Yaskawa INFORM job: SKRZYNIA_4640_-90_STOPNI_20BR.JBI

/JOB
//NAME SKRZYNIA_4640_-90_STOPNI_20BR
///FOLDERNAME 02-SKRZYNIE_JOBS
//POS
///NPOS 581,581,0,37,0,0
///TOOL 0
///POSTYPE PULSE
///PULSE
C00000=0,-52280,40443,0,6876,0
C00001=-82314,-24956,17040,-59626,-27382,-6248
C00002=-93910,-8625,17040,-59626,-43355,-6248
C00003=-98846,-1061,-42166,-80308,-57081,16120
C00004=-100452,6057,-48127,-85711,-56704,21322
C00005=-95817,31791,-34187,-84788,-63710,26674
C00006=-95573,33077,-33257,-84645,-64023,26851
C00007=-94315,33778,-32137,-85160,-63467,26714
C00008=-95573,33077,-33257,-84645,-64023,26851
C00009=-94948,31301,-36075,-85235,-63717,27152
C00010=-95573,33077,-33257,-84645,-64023,26851
C00011=-95263,33142,-33256,-84677,-63995,26850
C00012=-95263,33142,-33256,-84677,-63995,26850
C00013=-94230,33719,-32331,-85099,-63538,26735
C00014=-95263,33142,-33256,-84677,-63995,26850
C00015=-94794,31816,-35365,-85120,-63763,27076
C00016=-95263,33142,-33256,-84677,-63995,26850
C00017=-95260,33144,-33256,-84678,-63995,26850
C00018=-95260,33144,-33256,-84678,-63995,26850
C00019=-94260,33701,-32361,-85086,-63552,26738
C00020=-95738,35616,-30155,-83417,-65710,26451
C00021=-94835,31943,-35167,-85080,-63786,27056
C00022=-95260,33144,-33256,-84678,-63995,26850
C00023=-95258,25631,32269,-66559,-75499,2416
C00024=-95258,25631,32269,-66559,-75499,2416
C00025=-94256,26435,33444,-66420,-74940,2208
C00026=-95258,25631,32269,-66559,-75499,2416
C00027=-94857,24030,29962,-66606,-75105,2539
C00028=-95258,25631,32269,-66559,-75499,2416
C00029=-98811,21047,-15512,-99242,-81394,20987
C00030=-98811,21047,-15512,-99242,-81394,20987
C00031=-97856,21592,-14760,-99539,-80803,20995
C00032=-98811,21047,-15512,-99242,-81394,20987
C00033=-98487,19855,-17143,-99373,-81250,21110
C00034=-98811,21047,-15512,-99242,-81394,20987
C00035=-99077,36985,67047,-90824,-74996,11
C00036=-99077,36985,67047,-90824,-74996,11
C00037=-98126,38026,68808,-90519,-74354,-175
C00038=-99077,36985,67047,-90824,-74996,11
C00039=-98675,34279,62554,-90994,-74807,523
C00040=-99077,36985,67047,-90824,-74996,11
C00041=-98046,30065,45001,-99674,-75008,5996
C00042=-96663,27244,32711,-106417,-76052,10001
C00043=-96035,27733,33435,-106407,-75606,10011
C00044=-96663,27244,32711,-106417,-76052,10001
C00045=-96274,25568,30264,-106516,-75947,10234
C00046=-96663,27244,32711,-106417,-76052,10001
C00047=-100395,5963,-6492,-101051,-69866,13942
C00048=-97697,-21147,-29798,-104770,-52931,14344
C00049=-81691,-45027,-49520,-104186,-37412,14105
C00050=-48287,-44591,-17414,-16172,-14532,-25809
C00051=-85348,-13130,13838,-41209,-47455,-8220
C00052=-97998,22495,32685,-69647,-75009,8900
C00053=-98284,29564,37770,-71835,-80250,10571
C00054=-100615,26523,30326,-83718,-79542,3747
C00055=-99528,26746,30653,-83688,-78804,3698
C00056=-98609,27389,31597,-83640,-78189,3601
C00057=-99528,26746,30653,-83688,-78804,3698
C00058=-99278,25562,28929,-83734,-78615,3833
C00059=-99528,26746,30653,-83688,-78804,3698
C00060=-97827,29852,38067,-72347,-79830,10157
C00061=-97362,30289,38867,-71738,-79704,10396
C00062=-96447,31020,39967,-71637,-79179,10220
C00063=-97362,30289,38867,-71738,-79704,10396
C00064=-97069,28896,36765,-71776,-79401,10550
C00065=-97362,30289,38867,-71738,-79704,10396
C00066=-99687,30516,41738,-96594,-77984,-2813
C00067=-99279,34023,49568,-96204,-78485,-4167
C00068=-98297,34881,50932,-96068,-77785,-4257
C00069=-99279,34023,49568,-96204,-78485,-4167
C00070=-98948,32155,46632,-96284,-78364,-3863
C00071=-99279,34023,49568,-96204,-78485,-4167
C00072=-99820,26032,21623,-82067,-78848,-4447
C00073=-99820,26032,21623,-82067,-78848,-4447
C00074=-98898,26645,22513,-82083,-78237,-4546
C00075=-99820,26032,21623,-82067,-78848,-4447
C00076=-99438,24292,19129,-82156,-78552,-4268
C00077=-99820,26032,21623,-82067,-78848,-4447
C00078=-95331,1432,-9864,-84798,-60031,-3557
C00079=-100799,20404,12473,-99797,-78179,2590
C00080=-99814,-4938,-36996,-116444,-71342,12229
C00081=-82620,-30758,-83593,-142203,-62652,21635
C00082=-79591,-62427,-80212,-133576,-39445,13545
C00083=-61872,-66272,-83954,-148251,-32298,21081
C00084=-61872,-49557,-32264,-110357,-15428,1928
C00085=-71091,-37860,2722,-34648,-42002,-27792
C00086=-94097,-13222,20403,-45591,-54273,-19204
C00087=-97363,-23488,-17584,-60839,-44712,-9276
C00088=-98197,-8670,-25604,-81540,-55001,4479
C00089=-99236,18416,3235,-80713,-73731,6125
C00090=-98716,22747,8680,-80557,-75862,6048
C00091=-97982,23215,9333,-80619,-75386,5974
C00092=-98716,22747,8680,-80557,-75862,6048
C00093=-98409,21490,6932,-80649,-75627,6156
C00094=-98716,22747,8680,-80557,-75862,6048
C00095=-100183,29342,35466,-85708,-79719,1114
C00096=-100183,29342,35466,-85708,-79719,1114
C00097=-99011,30198,36753,-85631,-78926,990
C00098=-100183,29342,35466,-85708,-79719,1114
C00099=-99817,27493,32713,-85776,-79458,1347
C00100=-100183,29342,35466,-85708,-79719,1114
C00101=-94729,-288,3800,-87543,-55904,1533
C00102=-77861,-26606,-19905,-76223,-21443,-3330
C00103=-46440,-50562,-32626,1826,-13880,-39178
C00104=-46440,-50562,-32626,1826,-13880,-39178
///LIMIT ON
C00105=-38692,-65390,10180,-18335,3144,1955
///LIMIT OFF
C00106=0,-52280,40443,0,6876,0
C00107=0,-52280,40443,0,6876,0
C00108=0,-43112,23163,32261,-40956,29092
C00109=-48283,-21883,28214,-25170,-26491,48363
C00110=-46664,-3144,58041,-18842,-32105,45325
C00111=-50347,-18571,12268,-49104,-16423,60029
C00112=-52476,-17044,12146,-55476,-16783,62883
C00113=-51467,-16091,12918,-54586,-16145,62570
C00114=-51762,-16375,12685,-54854,-16332,62665
C00115=-53129,-15664,13268,-57063,-16995,63582
C00116=-52557,-17119,12084,-55547,-16837,62908
C00117=-50509,-19000,10610,-51503,-15997,61182
C00118=-52966,-16930,12240,-56194,-17032,63176
C00119=-51879,-15912,13067,-55265,-16346,62852
C00120=-52154,-16175,12851,-55507,-16521,62938
C00121=-53227,-15612,13314,-57215,-17042,63646
C00122=-52966,-16930,12240,-56194,-17032,63176
C00123=-50703,-18403,11066,-52155,-16024,61477
C00124=-52780,-17619,11680,-55562,-17015,62889
C00125=-51306,-16241,12790,-54268,-16084,62435
C00126=-51660,-16583,12512,-54593,-16308,62551
C00127=-53327,-15718,13220,-57282,-17114,63667
C00128=-52780,-17619,11680,-55562,-17015,62889
C00129=-50704,-18401,11069,-52157,-16021,61478
C00130=-53191,-17342,11901,-56260,-17204,63181
C00131=-51773,-16022,12969,-55050,-16305,62760
C00132=-52146,-16378,12679,-55379,-16540,62876
C00133=-53214,-15820,13135,-57085,-17059,63584
C00134=-53002,-17172,12037,-56105,-17083,63128
C00135=-51005,-17995,11387,-52847,-16122,61778
C00136=-52654,-17319,11922,-55560,-16911,62904
C00137=-51372,-16113,12897,-54432,-16099,62508
C00138=-51648,-16379,12679,-54684,-16273,62598
C00139=-52952,-15703,13233,-56807,-16903,63480
C00140=-53323,-17134,12070,-56539,-17248,63304
C00141=-52826,-20105,4812,-63938,-15678,66983
C00142=-52298,-19620,5183,-63681,-15322,66914
C00143=-51076,-18450,6096,-63049,-14499,66733
C00144=-51419,-18785,5831,-63233,-14731,66786
C00145=-52680,-18133,6347,-65138,-15424,67581
C00146=-52924,-19431,7025,-60935,-16175,65505
C00147=-51752,-18759,10786,-53484,-16613,62002
C00148=-52244,-17884,11471,-54682,-16766,62529
C00149=-50303,-16031,12961,-52880,-15542,61887
C00150=-50741,-16464,12607,-53310,-15818,62044
C00151=-52416,-15612,13306,-56135,-16617,63223
C00152=-51898,-18011,11369,-54129,-16600,62301
C00153=-50945,-18019,11363,-52741,-16103,61737
C00154=-51347,-17395,11856,-53690,-16237,62152
C00155=-49990,-16073,12923,-52376,-15383,61677
C00156=-50384,-16465,12603,-52769,-15629,61822
C00157=-52066,-15616,13298,-55654,-16423,63028
C00158=-51792,-17610,11685,-54205,-16494,62350
C00159=-50945,-18019,11363,-52741,-16103,61737
C00160=-50845,-17493,11778,-52895,-15987,61824
C00161=-49521,-16191,12826,-51571,-15155,61341
C00162=-49894,-16567,12520,-51958,-15389,61484
C00163=-51728,-15654,13268,-55171,-16246,62832
C00164=-51082,-17431,11827,-53280,-16102,61986
C00165=-50028,-23690,-6096,-22921,-31075,54538
C00166=-50346,-22995,-5584,-23393,-31002,54768
C00167=-48843,-21430,-4410,-21901,-30270,54078
C00168=-49178,-21788,-4683,-22239,-30433,54235
C00169=-50538,-21100,-4158,-23908,-30654,55032
C00170=-50252,-22811,-5450,-23315,-30936,54734
C00171=-49763,-24818,-32918,-23163,-28604,59699
C00172=-49144,-24298,-32242,-22455,-28505,59304
C00173=-47766,-22458,-30816,-21237,-27774,58615
C00174=-48099,-22913,-31171,-21534,-27949,58786
C00175=-49602,-21997,-30448,-23301,-28174,59772
C00176=-49259,-23869,-32392,-22880,-28141,59533
C00177=-50713,-12366,-58367,-41124,-17813,74400
C00178=-50097,-11438,-57505,-40749,-17495,74109
C00179=-49105,-9842,-55994,-40096,-16991,73614
C00180=-49355,-10250,-56383,-40269,-17116,73742
C00181=-50506,-9357,-55529,-41571,-17503,74586
C00182=-49771,-10920,-57018,-40545,-17327,73951
C00183=-46548,-30139,-39639,-20061,-27197,57955
C00184=-48797,-26670,-6576,-20404,-32539,53259
C00185=-45389,-28224,4312,-35967,-15579,54278
C00186=-40154,-51179,-915,-24203,-8234,36524
C00187=0,-52280,40443,0,6876,0
C00188=0,-52280,40443,0,6876,0
C00189=-2117,-50103,-33543,-4117,45077,85249
C00190=26439,-48928,-33543,-4117,-52362,85249
C00191=26439,-27355,-33543,-41485,-52362,85249
C00192=39218,-24492,-41653,-51934,-39374,86964
C00193=38244,-2284,-24157,-56964,-37300,90090
C00194=26640,586,-20198,-77712,-51919,89712
C00195=26323,460,-20341,-77681,-52125,89737
C00196=25607,3186,-17293,-77585,-52601,89760
C00197=26323,460,-20341,-77681,-52125,89737
C00198=27719,1044,-19697,-77798,-51218,89644
C00199=26640,586,-20198,-77712,-51919,89712
C00200=46457,7101,-11330,-26648,-40775,82885
C00201=47439,8350,-9833,-26106,-40556,82449
C00202=46334,10684,-6981,-26557,-41070,82837
C00203=47439,8350,-9833,-26106,-40556,82449
C00204=48354,9159,-8854,-25603,-40343,82046
C00205=47439,8350,-9833,-26106,-40556,82449
C00206=24760,-3019,-10726,-94610,-54398,89614
C00207=25145,-1220,-8811,-94681,-54143,89655
C00208=24492,1290,-6066,-94601,-54582,89624
C00209=25145,-1220,-8811,-94681,-54143,89655
C00210=26584,-669,-8211,-94866,-53174,89734
C00211=25145,-1220,-8811,-94681,-54143,89655
C00212=14532,-15164,-22494,-92943,-61192,88617
C00213=-33377,-12679,-20251,-90012,-93751,87621
C00214=-32674,-7309,22058,-70557,-98373,80594
C00215=20046,-29908,-41690,-58842,-55822,75080
C00216=46158,10269,-6164,-23128,-46470,70172
C00217=51306,10256,-19432,-23475,-33025,71236
C00218=50386,12004,-17260,-23922,-33430,71616
C00219=51306,10256,-19432,-23475,-33025,71236
C00220=51995,10928,-18601,-23012,-32906,70879
C00221=51306,10256,-19432,-23475,-33025,71236
C00222=50667,8104,-22050,-23976,-33027,71608
C00223=27434,3323,14960,-56922,-57501,78346
C00224=29014,6574,18756,-56344,-56678,77965
C00225=28326,9009,21700,-56459,-57175,78009
C00226=29014,6574,18756,-56344,-56678,77965
C00227=30292,7183,19486,-55908,-55969,77693
C00228=29014,6574,18756,-56344,-56678,77965
C00229=24457,-1296,-8898,-94600,-54606,89622
C00230=24457,-1296,-8898,-94600,-54606,89622
C00231=23939,748,-6672,-94541,-54956,89598
C00232=24457,-1296,-8898,-94600,-54606,89622
C00233=25626,-864,-8432,-94748,-53818,89684
C00234=24457,-1296,-8898,-94600,-54606,89622
C00235=22058,-20035,-26567,-93333,-56013,88551
C00236=-28907,-25632,-31027,-90338,-90583,86609
C00237=-23923,-11573,-19230,-90501,-87328,87840
C00238=-8646,-8251,-7782,-76032,-82054,83740
C00239=42001,26537,64712,-25019,-74648,68382
C00240=42692,25604,59505,-25067,-71864,68798
C00241=42100,27723,62792,-25233,-72628,68820
C00242=42692,25604,59505,-25067,-71864,68798
C00243=43179,26157,60355,-24838,-71882,68629
C00244=42692,25604,59505,-25067,-71864,68798
C00245=42064,17796,48100,-25604,-70267,69397
C00246=28113,-7386,-15136,-95790,-47335,90009
C00247=28228,-6488,-14240,-95859,-47266,90053
C00248=27767,-5044,-12775,-95858,-47588,90072
C00249=28228,-6488,-14240,-95859,-47266,90053
C00250=29468,-5989,-13737,-96077,-46438,90154
C00251=28228,-6488,-14240,-95859,-47266,90053
C00252=51937,664,-7429,-160484,-50080,89770
C00253=52345,1107,-6938,-160727,-50007,89930
C00254=51359,2767,-5080,-160136,-50147,89540
C00255=52345,1107,-6938,-160727,-50007,89930
C00256=53054,1752,-6222,-161147,-49882,90209
C00257=52345,1107,-6938,-160727,-50007,89930
C00258=51937,664,-7429,-160484,-50080,89770
C00259=29691,-10745,-18393,-95770,-46230,89933
C00260=26663,-19279,-25970,-94307,-48104,89008
C00261=29542,-7588,-14846,-100915,-46930,90773
C00262=29616,-6902,-10165,-96183,-45225,84004
C00263=29097,-5391,-8640,-96201,-45588,84023
C00264=29616,-6902,-10165,-96183,-45225,84004
C00265=31098,-6282,-9543,-96410,-44233,84135
C00266=29616,-6902,-10165,-96183,-45225,84004
C00267=7576,-30273,-44451,-97512,-61182,86443
C00268=-18624,-40022,-50597,-93591,-78329,83668
C00269=-32134,-30783,-37092,-96173,-88064,83581
C00270=23774,-1324,-8929,-94512,-55065,89585
C00271=23774,-1324,-8929,-94512,-55065,89585
C00272=23319,517,-6924,-94461,-55372,89567
C00273=23774,-1324,-8929,-94512,-55065,89585
C00274=25077,-853,-8421,-94674,-54188,89653
C00275=23774,-1324,-8929,-94512,-55065,89585
C00276=22107,-1052,28039,-94807,-51389,77849
C00277=19995,-16885,24938,-75612,-39910,62837
C00278=5366,-38499,37552,-33963,-10211,16191
C00279=0,-52280,40443,0,6876,0
C00280=-82314,-24956,17040,-59626,-27382,-6248
C00281=-93910,-8625,17040,-59626,-43355,-6248
C00282=-98846,-1061,-42166,-80308,-57081,16120
C00283=-100452,6057,-48127,-85711,-56704,21322
C00284=-95564,34698,-34234,-85516,-63941,27819
C00285=-94021,36658,-30981,-84167,-64832,27454
C00286=-93851,36773,-30815,-84181,-64812,27439
C00287=-95564,34698,-34234,-85516,-63941,27819
C00288=-96930,32282,-32252,-82595,-65816,26305
C00289=-93901,32995,-31122,-83953,-64436,26132
C00290=-93891,32978,-31150,-83961,-64431,26134
C00291=-96930,32282,-32252,-82595,-65816,26305
C00292=-97719,-4194,-31542,-76086,-54596,10626
C00293=-88377,-34186,-45291,-67238,-52212,2442
C00294=-73560,-62084,7826,-28695,-34737,-3666
C00295=0,-52280,40443,0,6876,0
C00296=0,-52280,40443,0,6876,0
C00297=-2117,-50103,-33543,-4117,45077,85249
C00298=26439,-48928,-33543,-4117,-52362,85249
C00299=26439,-27355,-33543,-41485,-52362,85249
C00300=39218,-24492,-41653,-51934,-39374,86964
C00301=37381,-5106,-22608,-53943,-39515,88347
C00302=38119,-10689,-19379,-70548,-34101,88029
C00303=37906,-14512,-22901,-69984,-34376,87713
C00304=41414,6981,-5927,-33889,-45598,86373
C00305=42289,10624,-1511,-33365,-45508,85956
C00306=42351,10656,-1473,-33340,-45486,85935
C00307=41414,6981,-5927,-33889,-45598,86373
C00308=53221,-12364,-8957,-19277,-47766,73858
C00309=11365,-15171,10010,-30164,-77975,82960
C00310=16156,-38280,11293,-23671,-42998,42040
C00311=11365,-47379,10010,-30164,3063,681
C00312=0,-52280,40443,0,6876,0
C00313=0,-36700,24612,42871,-31823,33862
C00314=-44403,-30110,7154,-24155,-23805,45557
C00315=-51570,-19542,10947,-41619,-21811,53396
C00316=-51570,-17239,16856,-38066,-23574,51584
C00317=-55052,-13712,19754,-43494,-24529,53873
C00318=-55190,-12778,21730,-42693,-25060,53437
C00319=-40431,-28773,9158,-17648,-23273,42875
C00320=0,-36700,24612,42871,-31823,33862
C00321=0,-52280,40443,0,6876,0
C00322=0,-52280,40443,0,6876,0
C00323=-73560,-62084,7826,-28695,-34737,-3666
C00324=-88377,-34186,-45291,-67238,-52212,2442
C00325=-99860,-8392,-35780,-75647,-56000,10650
C00326=-100432,21324,12575,-83706,-77956,7498
C00327=-100432,21324,12575,-83706,-77956,7498
C00328=-97477,24790,17443,-83584,-77881,7143
C00329=-97548,25214,18044,-83537,-78171,7107
C00330=-100432,21324,12575,-83706,-77956,7498
C00331=-100473,21504,12824,-83696,-77986,7482
C00332=-97708,25565,18549,-83502,-78342,7077
C00333=-97720,26100,19317,-83456,-78605,7025
C00334=-100432,21324,12575,-83706,-77956,7498
C00335=-98403,3681,-8965,-86029,-63956,7946
C00336=-99524,-11453,-5366,-86029,-50962,7946
C00337=-93426,-21174,-16075,-79197,-62083,2349
C00338=-58820,-39124,10926,-53325,-41870,-3759
C00339=0,-52280,40443,0,6876,0
C00340=-37281,-50778,-9546,-79570,-75313,71156
C00341=-21038,-23698,-30323,-82948,-81132,85647
C00342=-21230,-24252,-33397,-84866,-81311,86227
C00343=26224,-11477,-22521,-89106,-49066,87170
C00344=30473,789,4724,-68168,-47848,79016
C00345=30460,-1091,-3608,-71823,-46530,81583
C00346=26224,-11477,-22521,-89106,-49066,87170
C00347=1250,-26379,-34995,-85812,-66036,85728
C00348=-29373,-17697,-13794,-84248,-87305,82376
C00349=-12562,-22815,-22029,-52123,-75138,85349
C00350=41964,2536,-13642,-34848,-42769,74522
C00351=37974,4101,-26304,-58477,-36842,84551
C00352=37992,4823,-31618,-63468,-34913,87461
C00353=41439,5489,-14791,-37032,-40569,75962
C00354=38833,-3286,10682,-41231,-51577,69207
C00355=-9276,-22918,-17698,-90837,-69000,78700
C00356=-8172,-56778,-49528,-75726,-40055,75711
C00357=-3982,-61001,-53003,-69042,-33087,73336
C00358=37287,-55159,35520,-2191,5667,2084
C00359=0,-52280,40443,0,6876,0
C00360=0,-36700,24612,42871,-31823,33862
C00361=-44403,-30110,7154,-24155,-23805,45557
C00362=-44403,-30110,7154,-24155,-23805,45557
C00363=-42101,-12213,25656,-103795,-5192,78630
C00364=-46259,-8171,27719,-110365,-8144,81138
C00365=-49067,-3914,32085,-108223,-9817,79727
C00366=-55938,-2414,24284,-132193,-25662,89374
C00367=-55845,-2055,25408,-131547,-25258,89050
C00368=-56934,-15752,2926,-132390,-27589,90381
C00369=-47073,-34549,9488,-27883,-30316,51458
C00370=0,-52280,40443,0,6876,0
C00371=0,-52280,40443,0,6876,0
C00372=-73560,-62084,7826,-28695,-34737,-3666
C00373=-96366,-17217,16860,-56620,-71703,-18245
C00374=-98152,-14905,2044,-65675,-67485,-3494
C00375=-100467,-7393,-15195,-81625,-60158,6002
C00376=-99336,18440,8642,-84276,-74234,7647
C00377=-99336,18440,8642,-84276,-74234,7647
C00378=-97907,25479,18429,-83510,-78268,7080
C00379=-97774,25771,18838,-83486,-78362,7054
C00380=-99336,18440,8642,-84276,-74234,7647
C00381=-88887,-29565,-44699,-91336,-36715,8429
C00382=-85230,-48302,-58733,-86716,-36654,5475
C00383=-60204,-59872,-73451,-117647,-17639,18840
C00384=-37721,-67612,11381,-1325,-438,-7850
C00385=0,-52280,40443,0,6876,0
C00386=37287,-55159,35520,-2191,5667,2084
C00387=40042,-68802,-18337,-47708,-19461,45384
C00388=16481,-63411,-38742,-86271,-37962,67106
C00389=28646,-23138,-32952,-89786,-42552,85395
C00390=38882,-16596,-17625,-44304,-41043,72768
C00391=40930,-6862,-13364,-47045,-37020,74415
C00392=41744,-3361,-9781,-46774,-36492,74231
C00393=41678,-4243,-16493,-50979,-33997,76666
C00394=40930,-6862,-13364,-47045,-37020,74415
C00395=38882,-16596,-17625,-44304,-41043,72768
C00396=28646,-23138,-32952,-89786,-42552,85395
C00397=29905,-15291,-26411,-91102,-43435,86304
C00398=31540,-7654,-19248,-92177,-42391,86919
C00399=31445,-8095,-22888,-97196,-43117,89457
C00400=29637,-16450,-35189,-96198,-44206,89682
C00401=-7164,-46429,-55577,-86274,-68578,84143
C00402=40042,-68802,-18337,-47708,-19461,45384
C00403=37287,-55159,35520,-2191,5667,2084
C00404=0,-52280,40443,0,6876,0
C00405=-37164,-60659,6466,-13301,-5027,19773
C00406=-45362,-39990,2831,-27538,-17767,40935
C00407=-57189,-26834,-7130,-38780,-31731,51561
C00408=-55974,-20661,-3180,-39617,-29741,52134
C00409=-55991,-28453,-45977,-64163,-20900,63765
C00410=-57189,-26834,-7130,-38780,-31731,51561
C00411=-41180,-61187,4729,-17280,-8498,23442
C00412=0,-52280,40443,0,6876,0
C00413=0,-52280,40443,0,6876,0
C00414=-43180,-50572,-20637,-6552,-29302,-38834
C00415=-79425,-37128,-15462,-51820,-35721,-18807
C00416=-93702,-21743,-5664,-65079,-41536,-12324
C00417=-95468,-3718,3432,-57810,-54196,-8058
C00418=-98195,18244,29331,-65465,-72367,-4307
C00419=-96728,36447,56610,-70336,-82085,-4645
C00420=-96821,31985,42520,-71106,-80277,-1800
C00421=-99571,23446,29328,-71481,-76214,-993
C00422=-98368,-15155,-15320,-68503,-52006,-4003
C00423=-90196,-30440,-22000,-63685,-45526,-9297
C00424=-44920,-50063,-20090,-8739,-29356,-37564
C00425=-37721,-67612,11381,-1325,-438,-7850
C00426=0,-52280,40443,0,6876,0
C00427=40043,-68802,-18337,-47706,-19461,45383
C00428=27078,-46675,7729,-35821,-60236,53359
C00429=37661,6027,34279,-36092,-58837,68690
C00430=38848,9668,32452,-36978,-55195,69693
C00431=45203,15557,41040,-24527,-60177,66840
C00432=37661,2340,23735,-37788,-55306,70200
C00433=22173,-30639,7984,-58136,-45615,60133
C00434=37287,-55159,35520,-2191,5667,2084
C00435=0,-52280,40443,0,6876,0
C00436=-23708,-46776,23536,-16027,-4787,19738
C00437=-50917,-40459,4132,-34421,-18173,42391
C00438=-54964,-26842,8528,-44141,-23181,52038
C00439=-51719,-20944,8196,-48593,-18539,54728
C00440=-53338,-16066,12564,-52314,-18938,56375
C00441=-53668,-14237,17353,-48629,-20286,54493
C00442=-18010,-41727,-5437,24633,-20435,23511
C00443=-41180,-61187,4729,-17280,-8498,23442
C00444=0,-52280,40443,0,6876,0
C00445=0,-52280,40443,0,6876,0
C00446=-37721,-67612,11381,-1325,-438,-7850
C00447=-43180,-50572,-20637,-6552,-29302,-38834
C00448=-79425,-37128,-15462,-51820,-35721,-18807
C00449=-92377,-33385,-41303,-83059,-36844,-1354
C00450=-98043,-4314,-16897,-86107,-58749,2387
C00451=-99186,-1007,-13605,-90357,-63007,3800
C00452=-99448,23410,16807,-87478,-77479,2357
C00453=-98529,24761,18725,-87324,-78429,2215
C00454=-98419,25196,20150,-87169,-78534,1864
C00455=-99450,-173,-12700,-90327,-63185,3798
C00456=-99875,3426,-9244,-98609,-66692,6315
C00457=-99431,-3293,-16601,-99643,-62713,6757
C00458=-92822,-26306,-37175,-103295,-43881,7703
C00459=-68601,-52593,-52127,-95725,-25602,3235
C00460=-80632,-38079,-20908,-64053,-45216,-12949
C00461=-43180,-50572,-20637,-6552,-29302,-38834
C00462=-37721,-67612,11381,-1325,-438,-7850
C00463=0,-52280,40443,0,6876,0
C00464=-7830,-25136,17099,-55306,-64068,52084
C00465=34592,-23156,18291,-29932,-45204,43222
C00466=27626,-5609,7480,-74303,-46810,69713
C00467=30162,-7263,-3756,-79871,-43922,73611
C00468=30945,-3557,12,-79972,-43367,73694
C00469=30934,-3652,-86,-79966,-43372,73693
C00470=29106,-7674,-4162,-79972,-44640,73655
C00471=-2837,-32019,-23857,-80741,-66785,72567
C00472=9534,-43450,13514,-26959,-29486,38723
C00473=22834,-59963,22946,-6692,-2150,9612
C00474=0,-52280,40443,0,6876,0
C00475=-23708,-46776,23536,-16027,-4787,19738
C00476=-50917,-40459,4132,-34421,-18173,42391
C00477=-51059,-36587,4608,-36647,-19418,45358
C00478=-50113,-22729,10834,-36393,-23396,50963
C00479=-58003,-17258,7975,-66354,-22196,69294
C00480=-57660,-15851,11780,-61832,-22634,66694
C00481=-50113,-22729,10834,-36393,-23396,50963
C00482=-45969,-44671,-42317,80322,10570,10889
C00483=-31285,-69981,-10849,-7246,-6842,20992
C00484=0,-52280,40443,0,6876,0
C00485=-37721,-67612,11381,-1325,-438,-7850
C00486=-43180,-50572,-20637,-6552,-29302,-38834
C00487=-79425,-37128,-15462,-51820,-35721,-18807
C00488=-92377,-33385,-41303,-83059,-36844,-1354
C00489=-97955,-4566,-17156,-86109,-58691,2381
C00490=-98763,-4191,-27333,-97091,-62203,7437
C00491=-100541,17285,32324,-96596,-68502,-4435
C00492=-99163,31411,54049,-96228,-73919,-6997
C00493=-97653,31369,46884,-97568,-75920,-4787
C00494=-97653,34871,57346,-96543,-75121,-6929
C00495=-98792,6748,2422,-99606,-66785,1957
C00496=-99852,25442,19906,-82977,-78439,1439
C00497=-97669,24909,7904,-99153,-81388,7704
C00498=-97669,24909,7904,-99153,-81388,7704
C00499=-99984,22604,5279,-91306,-78940,6306
C00500=-98813,-5502,-22210,-93134,-60245,5727
C00501=-97559,-25159,-36085,-93407,-46496,3918
C00502=-68601,-52593,-52127,-95725,-25602,3235
C00503=-80632,-38079,-20908,-64053,-45216,-12949
C00504=-43180,-50572,-20637,-6552,-29302,-38834
C00505=-37721,-67612,11381,-1325,-438,-7850
C00506=54026,-30203,28811,7745,-28969,5087
C00507=55906,-29650,27841,6704,-28568,42061
C00508=3910,-49110,-20873,-64325,-51391,71742
C00509=9596,-41005,-15480,-61992,-50741,70573
C00510=34629,-5327,8260,-51720,-47880,65426
C00511=35679,2837,17551,-51053,-47466,65038
C00512=35689,-56,7549,-54586,-44718,67469
C00513=34629,-5327,8260,-51720,-47880,65426
C00514=9596,-41005,-15480,-61992,-50741,70573
C00515=29660,-4584,-26917,-122917,-59269,85605
C00516=30458,-1431,-23593,-123278,-58903,85810
C00517=32051,-581,-21149,-126899,-58917,85995
C00518=28378,-5181,-30467,-124970,-61925,86269
C00519=9596,-41005,-15480,-61992,-50741,70573
C00520=4124,-42500,-16101,-63937,-54198,71061
C00521=22834,-59963,22946,-6692,-2150,9612
C00522=0,-52280,40443,0,6876,0
C00523=-44101,-76445,-48847,-15697,-17168,40457
C00524=-48984,-30078,-36716,-21434,-29637,58750
C00525=-50484,-13386,-55713,-36158,-19724,71897
C00526=-50484,-10141,-52609,-36672,-19476,72159
C00527=-57834,15023,-57436,-77444,-21310,89314
C00528=-50484,-13386,-55713,-36158,-19724,71897
C00529=-49763,-25421,-36239,-24565,-26935,60445
C00530=-50529,-22709,-3778,-22940,-31995,54502
C00531=-45389,-28224,4312,-35967,-15579,54278
C00532=-40154,-51179,-915,-24203,-8234,36524
C00533=0,-52280,40443,0,6876,0
C00534=0,-52280,40443,0,6876,0
C00535=-37721,-67612,11381,-1325,-438,-7850
C00536=-43180,-50572,-20637,-6552,-29302,-38834
C00537=-43180,-50572,-20637,-6552,-29302,-38834
C00538=-91571,-17240,10754,-52986,-45776,-17944
C00539=-85565,-2479,24798,-50710,-47830,-17652
C00540=-84901,-1641,24348,-52361,-47087,-17020
C00541=-100018,24469,26124,-84922,-77496,-993
C00542=-98221,24171,26084,-84881,-76275,-1110
C00543=-97925,23780,23736,-81145,-76027,-1196
C00544=-96886,22779,17134,-75074,-74614,-730
C00545=-96886,21697,9827,-76119,-73731,1247
C00546=-99355,23812,23162,-76774,-76908,-1703
C00547=-99772,22813,18672,-85812,-76963,849
C00548=-98588,26860,21106,-87462,-79585,-1754
C00549=-98621,27173,20618,-87985,-79896,-2348
C00550=-99360,20896,24116,-84704,-74336,-1671
C00551=-89794,-9992,-7341,-81590,-44258,-3681
C00552=-98228,-14972,-11291,-81392,-49231,-4002
C00553=-98228,-7428,13566,-72439,-51372,-10695
C00554=-68865,-35989,-5252,-49829,-38105,-21179
C00555=-40763,-44623,-7750,-16844,-36810,-34738
C00556=0,-52278,40443,-31822,-65283,46097
C00557=7820,3000,44222,-77356,-66876,70486
C00558=23103,22769,71034,-65639,-61603,67373
C00559=25078,30713,84198,-63240,-61811,65668
C00560=25008,30264,83410,-63369,-61766,65773
C00561=23103,22769,71034,-65639,-61603,67373
C00562=23103,22769,71034,-65639,-61603,67373
C00563=25078,30713,84198,-63240,-61811,65668
C00564=25008,30264,83410,-63369,-61766,65773
C00565=23103,22769,71034,-65639,-61603,67373
C00566=-3014,-20441,-7349,-104591,-68614,79454
C00567=-3014,-20441,-7349,-104591,-68614,79454
C00568=-13238,-21720,-1359,-93359,-59492,72612
C00569=10261,-46634,14475,-36899,-22136,31570
C00570=22834,-59963,22946,-6692,-2150,9612
C00571=0,-52280,40443,0,6876,0
C00572=-23708,-46776,23536,-16027,-4787,19738
C00573=-50917,-40459,4132,-34421,-18173,42391
C00574=-49876,-21948,7530,-68838,-10324,59148
C00575=-46721,-18942,9765,-68167,-8197,59205
C00576=-47734,-15041,12007,-78406,-8476,63945
C00577=-48173,-14749,12492,-78097,-8776,63748
C00578=-42573,-24036,4541,-56448,-5917,54155
C00579=-31287,-69981,-10850,-7253,-6843,20996
C00580=0,-52280,40443,0,6876,0
BC00000=455888
BC00001=445130
BC00002=445130
BC00003=445130
BC00004=445130
BC00005=467179
BC00006=468227
BC00007=468227
BC00008=468227
BC00009=468227
BC00010=468227
BC00011=514421
BC00012=514421
BC00013=514421
BC00014=514421
BC00015=514421
BC00016=514421
BC00017=560588
BC00018=560588
BC00019=560588
BC00020=560588
BC00021=560588
BC00022=560588
BC00023=536404
BC00024=536404
BC00025=536404
BC00026=536404
BC00027=536404
BC00028=536404
BC00029=582458
BC00030=582458
BC00031=582458
BC00032=582458
BC00033=582458
BC00034=582458
BC00035=581206
BC00036=581206
BC00037=581206
BC00038=581206
BC00039=581206
BC00040=581206
BC00041=608443
BC00042=608308
BC00043=608308
BC00044=608308
BC00045=608308
BC00046=608308
BC00047=554082
BC00048=550688
BC00049=540680
BC00050=699121
BC00051=714117
BC00052=772491
BC00053=770398
BC00054=668005
BC00055=668005
BC00056=668005
BC00057=668005
BC00058=668005
BC00059=668005
BC00060=765624
BC00061=770398
BC00062=770398
BC00063=770398
BC00064=770398
BC00065=770398
BC00066=795066
BC00067=795066
BC00068=795066
BC00069=795066
BC00070=795066
BC00071=795066
BC00072=855510
BC00073=855510
BC00074=855510
BC00075=855510
BC00076=855510
BC00077=855510
BC00078=855510
BC00079=800260
BC00080=807414
BC00081=829241
BC00082=831883
BC00083=872244
BC00084=872244
BC00085=900921
BC00086=897901
BC00087=922181
BC00088=915260
BC00089=906767
BC00090=899976
BC00091=899976
BC00092=899976
BC00093=899976
BC00094=899976
BC00095=940845
BC00096=940845
BC00097=940845
BC00098=940845
BC00099=940845
BC00100=940845
BC00101=861557
BC00102=891834
BC00103=895420
BC00104=874556
BC00105=799329
BC00106=750352
BC00107=750350
BC00108=750352
BC00109=858258
BC00110=858258
BC00111=887560
BC00112=953382
BC00113=953382
BC00114=953382
BC00115=953382
BC00116=953382
BC00117=888056
BC00118=888056
BC00119=888056
BC00120=888056
BC00121=888056
BC00122=888056
BC00123=830714
BC00124=830714
BC00125=830714
BC00126=830714
BC00127=830714
BC00128=830714
BC00129=764829
BC00130=764829
BC00131=764829
BC00132=764829
BC00133=764829
BC00134=764829
BC00135=707174
BC00136=707174
BC00137=707174
BC00138=707174
BC00139=707174
BC00140=707174
BC00141=642071
BC00142=642071
BC00143=642071
BC00144=642071
BC00145=642071
BC00146=642071
BC00147=584746
BC00148=584746
BC00149=584746
BC00150=584746
BC00151=584746
BC00152=584746
BC00153=519232
BC00154=519232
BC00155=519232
BC00156=519232
BC00157=519232
BC00158=519232
BC00159=461813
BC00160=461813
BC00161=461813
BC00162=461813
BC00163=461813
BC00164=461813
BC00165=459544
BC00166=459544
BC00167=459544
BC00168=459544
BC00169=459544
BC00170=459544
BC00171=459544
BC00172=459544
BC00173=459544
BC00174=459544
BC00175=459544
BC00176=459544
BC00177=459544
BC00178=459544
BC00179=459544
BC00180=459544
BC00181=459544
BC00182=459544
BC00183=459544
BC00184=459544
BC00185=459540
BC00186=533216
BC00187=533216
BC00188=492150
BC00189=423885
BC00190=423885
BC00191=423885
BC00192=423885
BC00193=423885
BC00194=423882
BC00195=423882
BC00196=423882
BC00197=423882
BC00198=423882
BC00199=423882
BC00200=517447
BC00201=516208
BC00202=516208
BC00203=516208
BC00204=516208
BC00205=516208
BC00206=462401
BC00207=462401
BC00208=462401
BC00209=462401
BC00210=462401
BC00211=462401
BC00212=462401
BC00213=462401
BC00214=581968
BC00215=647467
BC00216=647467
BC00217=647467
BC00218=647467
BC00219=647467
BC00220=647467
BC00221=647467
BC00222=647467
BC00223=600589
BC00224=600589
BC00225=600589
BC00226=600589
BC00227=600589
BC00228=600589
BC00229=646713
BC00230=646713
BC00231=646713
BC00232=646713
BC00233=646713
BC00234=646713
BC00235=646713
BC00236=646713
BC00237=703926
BC00238=764819
BC00239=734650
BC00240=734650
BC00241=734650
BC00242=734650
BC00243=734650
BC00244=734650
BC00245=734650
BC00246=762000
BC00247=762000
BC00248=762000
BC00249=762000
BC00250=762000
BC00251=762000
BC00252=768744
BC00253=768744
BC00254=768744
BC00255=768744
BC00256=768744
BC00257=768744
BC00258=768744
BC00259=762000
BC00260=762000
BC00261=869424
BC00262=869424
BC00263=869424
BC00264=869424
BC00265=869424
BC00266=869424
BC00267=869424
BC00268=869424
BC00269=983898
BC00270=992364
BC00271=992364
BC00272=992364
BC00273=992364
BC00274=992364
BC00275=992364
BC00276=927243
BC00277=910363
BC00278=716208
BC00279=458496
BC00280=445130
BC00281=445130
BC00282=445130
BC00283=445130
BC00284=475938
BC00285=475917
BC00286=468314
BC00287=475938
BC00288=515329
BC00289=515329
BC00290=508301
BC00291=515329
BC00292=542207
BC00293=542207
BC00294=542207
BC00295=542207
BC00296=492150
BC00297=423885
BC00298=423885
BC00299=423885
BC00300=423885
BC00301=418215
BC00302=406365
BC00303=406365
BC00304=507950
BC00305=507950
BC00306=500226
BC00307=507950
BC00308=493160
BC00309=493160
BC00310=493160
BC00311=493160
BC00312=493160
BC00313=582810
BC00314=655182
BC00315=714528
BC00316=712780
BC00317=712780
BC00318=773753
BC00319=773753
BC00320=582810
BC00321=540924
BC00322=542207
BC00323=542207
BC00324=542207
BC00325=590944
BC00326=543764
BC00327=459277
BC00328=459277
BC00329=451665
BC00330=459277
BC00331=520748
BC00332=520748
BC00333=528295
BC00334=520748
BC00335=524597
BC00336=524597
BC00337=555662
BC00338=584417
BC00339=584417
BC00340=542360
BC00341=599440
BC00342=482963
BC00343=482963
BC00344=482963
BC00345=482963
BC00346=482963
BC00347=482963
BC00348=482963
BC00349=633179
BC00350=633182
BC00351=633182
BC00352=633182
BC00353=633182
BC00354=590162
BC00355=577838
BC00356=565789
BC00357=612529
BC00358=620193
BC00359=620193
BC00360=812803
BC00361=887783
BC00362=927066
BC00363=893694
BC00364=914884
BC00365=914884
BC00366=943670
BC00367=973194
BC00368=945981
BC00369=853059
BC00370=542207
BC00371=542207
BC00372=513519
BC00373=556866
BC00374=576802
BC00375=590944
BC00376=571989
BC00377=566860
BC00378=566866
BC00379=572997
BC00380=566860
BC00381=580682
BC00382=599892
BC00383=633159
BC00384=733103
BC00385=733103
BC00386=620193
BC00387=620193
BC00388=625652
BC00389=635598
BC00390=635598
BC00391=635598
BC00392=635598
BC00393=635598
BC00394=635598
BC00395=635598
BC00396=635598
BC00397=658627
BC00398=658630
BC00399=665879
BC00400=658627
BC00401=658627
BC00402=620193
BC00403=620193
BC00404=620193
BC00405=561542
BC00406=498768
BC00407=452071
BC00408=452071
BC00409=452071
BC00410=452071
BC00411=524165
BC00412=524165
BC00413=733103
BC00414=733103
BC00415=646139
BC00416=646133
BC00417=684512
BC00418=682982
BC00419=682982
BC00420=682982
BC00421=682982
BC00422=682236
BC00423=687704
BC00424=698572
BC00425=733103
BC00426=733103
BC00427=667407
BC00428=721208
BC00429=721208
BC00430=721208
BC00431=727232
BC00432=730010
BC00433=686453
BC00434=620193
BC00435=620193
BC00436=576077
BC00437=541793
BC00438=580754
BC00439=589556
BC00440=589433
BC00441=647350
BC00442=649294
BC00443=561088
BC00444=547800
BC00445=733103
BC00446=733103
BC00447=733103
BC00448=733103
BC00449=733103
BC00450=733103
BC00451=740531
BC00452=740531
BC00453=740531
BC00454=745553
BC00455=740531
BC00456=750469
BC00457=750469
BC00458=750469
BC00459=750469
BC00460=783373
BC00461=795297
BC00462=733103
BC00463=733103
BC00464=727492
BC00465=727492
BC00466=759331
BC00467=759331
BC00468=759331
BC00469=766564
BC00470=759331
BC00471=759331
BC00472=672725
BC00473=672725
BC00474=672725
BC00475=766882
BC00476=791101
BC00477=802867
BC00478=836517
BC00479=836517
BC00480=895002
BC00481=836517
BC00482=798026
BC00483=767805
BC00484=733103
BC00485=733103
BC00486=733103
BC00487=733103
BC00488=733103
BC00489=733103
BC00490=815683
BC00491=777789
BC00492=777789
BC00493=784987
BC00494=784987
BC00495=788909
BC00496=855225
BC00497=846870
BC00498=855158
BC00499=855225
BC00500=811096
BC00501=804355
BC00502=750469
BC00503=783373
BC00504=795297
BC00505=733103
BC00506=762701
BC00507=765633
BC00508=830967
BC00509=835024
BC00510=852883
BC00511=852883
BC00512=852883
BC00513=852883
BC00514=835024
BC00515=861491
BC00516=861491
BC00517=861491
BC00518=861491
BC00519=835024
BC00520=835024
BC00521=672725
BC00522=672725
BC00523=528256
BC00524=459544
BC00525=459544
BC00526=459546
BC00527=459544
BC00528=459544
BC00529=459544
BC00530=459544
BC00531=459540
BC00532=533216
BC00533=533216
BC00534=733103
BC00535=733103
BC00536=854587
BC00537=886854
BC00538=885269
BC00539=885269
BC00540=923671
BC00541=946274
BC00542=946274
BC00543=946274
BC00544=907872
BC00545=907872
BC00546=907872
BC00547=970029
BC00548=970060
BC00549=977448
BC00550=970029
BC00551=911970
BC00552=906746
BC00553=883967
BC00554=913920
BC00555=863532
BC00556=921533
BC00557=921533
BC00558=946591
BC00559=946591
BC00560=953713
BC00561=946591
BC00562=997282
BC00563=997282
BC00564=1004404
BC00565=997282
BC00566=1013986
BC00567=963295
BC00568=908449
BC00569=754884
BC00570=672725
BC00571=672725
BC00572=562340
BC00573=452362
BC00574=452362
BC00575=452362
BC00576=452362
BC00577=512870
BC00578=511886
BC00579=742282
BC00580=742282
///POSTYPE BASE
///RECTAN
///RCONF 1,0,0,0,0,0,0,0,0,0,0,0,0,0,0,0,0,0,0,0,0,0,0,0
P00006=0.000,0.000,0.000,0.0000,0.0000,0.0000
P00300=-0.036,-1.505,2.318,0.0000,0.0000,0.0000
P00301=0.046,-2.112,7.779,0.0000,0.0000,0.0000
P00302=-0.180,-2.409,6.326,0.0000,0.0000,0.0000
///RCONF 0,0,0,0,0,0,0,0,0,0,0,0,0,0,0,0,0,0,0,0,0,0,0,0
P00303=-0.004,-1.437,-4.584,0.0000,0.0000,0.0000
P00304=0.028,-1.666,-4.234,0.0000,0.0000,0.0000
P00305=-0.003,-1.920,-3.501,0.0000,0.0000,0.0000
P00306=0.015,-2.252,-3.054,0.0000,0.0000,0.0000
P00307=0.019,-2.151,-5.077,0.0000,0.0000,0.0000
P00308=-0.003,-2.092,-4.888,0.0000,0.0000,0.0000
P00309=-0.040,-2.205,-4.992,0.0000,0.0000,0.0000
P00310=-0.006,-2.490,-5.925,0.0000,0.0000,0.0000
P00311=-0.007,-2.079,-5.307,0.0000,0.0000,0.0000
P00350=11.519,-0.008,1.149,0.0000,0.0000,0.0000
P00351=13.563,-0.027,-0.653,0.0000,0.0000,0.0000
P00352=13.252,-0.027,-0.827,0.0000,0.0000,0.0000
P00353=10.971,-0.082,0.776,0.0000,0.0000,0.0000
P00354=-0.024,2.508,-1.824,0.0000,0.0000,0.0000
P00355=-0.001,2.528,-1.131,0.0000,0.0000,0.0000
P00356=-0.034,2.921,-0.262,0.0000,0.0000,0.0000
P00357=0.003,3.386,-0.091,0.0000,0.0000,0.0000
P00358=0.014,3.037,-0.020,0.0000,0.0000,0.0000
P00359=-0.005,2.731,0.912,0.0000,0.0000,0.0000
P00360=-0.011,3.412,0.438,0.0000,0.0000,0.0000
P00361=0.018,3.050,1.253,0.0000,0.0000,0.0000
P00400=5.920,-3.503,-0.024,0.0000,0.0000,0.0000
P00401=3.430,-0.021,1.131,0.0000,0.0000,0.0000
P00402=-0.253,1.107,3.062,0.0000,0.0000,0.0000
P00403=-3.666,-0.015,5.328,0.0000,0.0000,0.0000
///RCONF 1,0,0,0,0,0,0,0,0,0,0,0,0,0,0,0,0,0,0,0,0,0,0,0
P00404=0.029,4.189,-1.030,0.0000,0.0000,0.0000
///RCONF 0,0,0,0,0,0,0,0,0,0,0,0,0,0,0,0,0,0,0,0,0,0,0,0
P00405=2.420,0.007,1.427,0.0000,0.0000,0.0000
P00406=3.513,-0.022,0.429,0.0000,0.0000,0.0000
///RCONF 1,0,0,0,1,0,0,0,0,0,0,0,0,0,0,0,0,0,0,0,0,0,0,0
P00407=-0.029,2.348,-1.469,0.0000,0.0000,0.0000
P00408=0.010,1.346,-1.479,0.0000,0.0000,0.0000
///RCONF 1,0,0,0,0,0,0,0,0,0,0,0,0,0,0,0,0,0,0,0,0,0,0,0
P00409=-0.026,2.090,-1.483,0.0000,0.0000,0.0000
P00410=0.001,4.491,-0.583,0.0000,0.0000,0.0000
///RCONF 1,0,0,0,1,0,0,0,0,0,0,0,0,0,0,0,0,0,0,0,0,0,0,0
P00411=-0.015,3.627,0.872,0.0000,0.0000,0.0000
//INST
///DATE 2024/11/22 15:59
///ATTR SC,RW
///GROUP1 RB1,BS1
NOP
CALL JOB:MOVE_INTO_TUNNEL
MOVJ C00000 BC00000 VJ=30.00
MOVJ C00001 BC00001 VJ=30.00
MOVJ C00002 BC00002 VJ=30.00
MOVL C00003 BC00003 V=500.0
MOVJ C00004 BC00004 VJ=20.00
'------------------------
'W65.3
'------------------------
MOVL C00005 BC00005 V=333.3
MOVL C00006 BC00006 V=166.7 PL=0
REFP 3 C00007 BC00007
CALL JOB:SEARCH-R1
SET P0300 P0006
SFTON P0300
MOVL C00008 BC00008 V=66.7 PL=0
REFP 3 C00009 BC00009
CALL JOB:SEARCH-R1
SET P0300 P0006
SFTON P0300
MOVL C00010 BC00010 V=66.7 PL=0
SFTOF
'------------------------
'W65.5
'------------------------
MOVL C00011 BC00011 V=500.0
MOVL C00012 BC00012 V=166.7 PL=0
REFP 3 C00013 BC00013
CALL JOB:SEARCH-R1
SET P0301 P0006
SFTON P0301
MOVL C00014 BC00014 V=166.7 PL=0
REFP 3 C00015 BC00015
CALL JOB:SEARCH-R1
SET P0301 P0006
SFTON P0301
MOVL C00016 BC00016 V=166.7 PL=0
SFTOF
'------------------------
'W65.7
'------------------------
MOVL C00017 BC00017 V=500.0
MOVL C00018 BC00018 V=166.7 PL=0
REFP 3 C00019 BC00019
CALL JOB:SEARCH-R1
SET P0302 P0006
SFTON P0302
MOVL C00020 BC00020 V=166.7 PL=0
REFP 3 C00021 BC00021
CALL JOB:SEARCH-R1
SET P0302 P0006
SFTON P0302
MOVL C00022 BC00022 V=166.7 PL=0
SFTOF
'------------------------
'W65.10
'------------------------
MOVL C00023 BC00023 V=500.0
MOVL C00024 BC00024 V=166.7 PL=0
REFP 3 C00025 BC00025
CALL JOB:SEARCH-R1
SET P0303 P0006
SFTON P0303
MOVL C00026 BC00026 V=166.7 PL=0
REFP 3 C00027 BC00027
CALL JOB:SEARCH-R1
SET P0303 P0006
SFTON P0303
MOVL C00028 BC00028 V=166.7 PL=0
SFTOF
'------------------------
'W65.12
'------------------------
MOVL C00029 BC00029 V=500.0
MOVL C00030 BC00030 V=166.7 PL=0
REFP 3 C00031 BC00031
CALL JOB:SEARCH-R1
SET P0304 P0006
SFTON P0304
MOVL C00032 BC00032 V=166.7 PL=0
REFP 3 C00033 BC00033
CALL JOB:SEARCH-R1
SET P0304 P0006
SFTON P0304
MOVL C00034 BC00034 V=166.7 PL=0
SFTOF
'------------------------
'W65.15
'------------------------
COMM MOVL C00035 BC00035 V=333.3
COMM MOVL C00036 BC00036 V=166.7 PL=0
COMM REFP 3 C00037 BC00037
COMM CALL JOB:SEARCH-R1
COMM SET P0305 P0006
COMM SFTON P0305
COMM MOVL C00038 BC00038 V=166.7 PL=0
COMM REFP 3 C00039 BC00039
COMM CALL JOB:SEARCH-R1
COMM SET P0305 P0006
COMM SFTON P0305
COMM MOVL C00040 BC00040 V=166.7 PL=0
COMM SFTOF
COMM '------------------------
COMM 'W65.17
COMM '------------------------
COMM MOVL C00041 BC00041 V=333.3
COMM MOVL C00042 BC00042 V=166.7 PL=0
COMM REFP 3 C00043 BC00043
COMM CALL JOB:SEARCH-R1
COMM SET P0306 P0006
COMM SFTON P0306
COMM MOVL C00044 BC00044 V=166.7 PL=0
COMM REFP 3 C00045 BC00045
COMM CALL JOB:SEARCH-R1
COMM SET P0306 P0006
COMM SFTON P0306
COMM MOVL C00046 BC00046 V=166.7 PL=0
COMM SFTOF
MOVL C00047 BC00047 V=333.3
MOVL C00048 BC00048 V=500.0
MOVL C00049 BC00049 V=500.0
MOVJ C00050 BC00050 VJ=50.00
MOVL C00051 BC00051 V=500.0
MOVL C00052 BC00052 V=500.0
'------------------------
'W65.20
'------------------------
MOVL C00053 BC00053 V=166.7
MOVL C00054 BC00054 V=416.7
MOVL C00055 BC00055 V=166.7 PL=0
REFP 3 C00056 BC00056
CALL JOB:SEARCH-R1
SET P0306 P0006
SFTON P0306
MOVL C00057 BC00057 V=166.7 PL=0
REFP 3 C00058 BC00058
CALL JOB:SEARCH-R1
SET P0306 P0006
SFTON P0306
MOVL C00059 BC00059 V=166.7 PL=0
SFTOF
MOVL C00060 BC00060 V=416.7
MOVL C00061 BC00061 V=166.7 PL=0
REFP 3 C00062 BC00062
CALL JOB:SEARCH-R1
SET P0307 P0006
SFTON P0307
MOVL C00063 BC00063 V=166.7 PL=0
REFP 3 C00064 BC00064
CALL JOB:SEARCH-R1
SET P0307 P0006
SFTON P0307
MOVL C00065 BC00065 V=166.7 PL=0
SFTOF
'------------------------
'W65.23
'------------------------
MOVL C00066 BC00066 V=333.3
MOVL C00067 BC00067 V=166.7 PL=0
REFP 3 C00068 BC00068
CALL JOB:SEARCH-R1
SET P0308 P0006
SFTON P0308
MOVL C00069 BC00069 V=166.7 PL=0
REFP 3 C00070 BC00070
CALL JOB:SEARCH-R1
SET P0308 P0006
SFTON P0308
MOVL C00071 BC00071 V=166.7 PL=0
SFTOF
'------------------------
'W65.25
'------------------------
COMM MOVL C00072 BC00072 V=500.0
COMM MOVL C00073 BC00073 V=166.7 PL=0
COMM REFP 3 C00074 BC00074
COMM CALL JOB:SEARCH-R1
COMM SET P0309 P0006
COMM SFTON P0309
COMM MOVL C00075 BC00075 V=166.7 PL=0
COMM REFP 3 C00076 BC00076
COMM CALL JOB:SEARCH-R1
COMM SET P0309 P0006
COMM SFTON P0309
COMM MOVL C00077 BC00077 V=166.7 PL=0
COMM SFTOF
COMM MOVL C00078 BC00078 V=166.7
MOVL C00079 BC00079 V=666.7
MOVL C00080 BC00080 V=666.7
MOVL C00081 BC00081 V=666.7
MOVL C00082 BC00082 V=666.7
MOVL C00083 BC00083 V=666.7
MOVL C00084 BC00084 V=666.7
MOVL C00085 BC00085 V=666.7
MOVL C00086 BC00086 V=666.7
MOVL C00087 BC00087 V=666.7
MOVL C00088 BC00088 V=500.0
MOVL C00089 BC00089 V=333.3
'------------------------
'W65.28
'------------------------
MOVL C00090 BC00090 V=166.7 PL=0
REFP 3 C00091 BC00091
CALL JOB:SEARCH-R1
SET P0310 P0006
SFTON P0310
MOVL C00092 BC00092 V=166.7 PL=0
REFP 3 C00093 BC00093
CALL JOB:SEARCH-R1
SET P0310 P0006
SFTON P0310
MOVL C00094 BC00094 V=166.7 PL=0
SFTOF
'------------------------
COMM 'W65.30
COMM '------------------------
COMM MOVL C00095 BC00095 V=500.0
COMM MOVL C00096 BC00096 V=166.7 PL=0
COMM REFP 3 C00097 BC00097
COMM CALL JOB:SEARCH-R1
COMM SET P0311 P0006
COMM SFTON P0311
COMM MOVL C00098 BC00098 V=166.7 PL=0
COMM REFP 3 C00099 BC00099
COMM CALL JOB:SEARCH-R1
COMM SET P0311 P0006
COMM SFTON P0311
COMM MOVL C00100 BC00100 V=166.7 PL=0
COMM SFTOF
MOVL C00101 BC00101 V=333.3
MOVL C00102 BC00102 V=333.3
MOVL C00103 BC00103 V=333.3
MOVL C00104 BC00104 V=666.7
MOVJ C00105 BC00105 VJ=50.00
MOVJ C00106 BC00106 VJ=50.00
MOVJ C00107 BC00107 VJ=10.00
MOVJ C00108 BC00108 VJ=50.00
MOVJ C00109 BC00109 VJ=30.00
MOVJ C00110 BC00110 VJ=30.00
MOVL C00111 BC00111 V=333.3
COMM SFTOF
COMM '------------------------
COMM 'W251A
COMM '------------------------
COMM MOVL C00112 BC00112 V=166.7 PL=0
COMM REFP 3 C00113 BC00113
COMM CALL JOB:SEARCH-R1
COMM SET P0350 P0006
COMM SFTON P0350
COMM MOVL C00114 BC00114 V=166.7 PL=0
COMM REFP 3 C00115 BC00115
COMM CALL JOB:SEARCH-R1
COMM SET P0350 P0006
COMM SFTON P0350
COMM MOVL C00116 BC00116 V=166.7 PL=0
SFTOF
'------------------------
'W254A P
'------------------------
MOVJ C00117 BC00117 VJ=40.00
MOVL C00118 BC00118 V=166.7 PL=0
REFP 3 C00119 BC00119
CALL JOB:SEARCH-R1
SET P0351 P0006
SFTON P0351
MOVL C00120 BC00120 V=166.7 PL=0
REFP 3 C00121 BC00121
CALL JOB:SEARCH-R1
SET P0351 P0006
SFTON P0351
MOVL C00122 BC00122 V=166.7 PL=0
SFTOF
'------------------------
'W254A L
'------------------------
MOVJ C00123 BC00123 VJ=40.00
MOVL C00124 BC00124 V=166.7 PL=0
REFP 3 C00125 BC00125
CALL JOB:SEARCH-R1
SET P0352 P0006
SFTON P0352
MOVL C00126 BC00126 V=166.7 PL=0
REFP 3 C00127 BC00127
CALL JOB:SEARCH-R1
SET P0352 P0006
SFTON P0352
MOVL C00128 BC00128 V=166.7 PL=0
SFTOF
'------------------------
'W250A P
'------------------------
MOVJ C00129 BC00129 VJ=40.00
MOVL C00130 BC00130 V=166.7 PL=0
REFP 3 C00131 BC00131
CALL JOB:SEARCH-R1
SET P0353 P0006
SFTON P0353
MOVL C00132 BC00132 V=66.7 PL=0
REFP 3 C00133 BC00133
CALL JOB:SEARCH-R1
SET P0353 P0006
SFTON P0353
MOVL C00134 BC00134 V=66.7 PL=0
SFTOF
'------------------------
'W250A L
'------------------------
MOVJ C00135 BC00135 VJ=40.00
MOVL C00136 BC00136 V=166.7 PL=0
REFP 3 C00137 BC00137
CALL JOB:SEARCH-R1
SET P0354 P0006
SFTON P0354
MOVL C00138 BC00138 V=66.7 PL=0
REFP 3 C00139 BC00139
CALL JOB:SEARCH-R1
SET P0354 P0006
SFTON P0354
MOVL C00140 BC00140 V=166.7 PL=0
SFTOF
'------------------------
'W253A P
'------------------------
MOVJ C00141 BC00141 VJ=40.00
MOVL C00142 BC00142 V=166.7 PL=0
REFP 3 C00143 BC00143
CALL JOB:SEARCH-R1
SET P0355 P0006
SFTON P0355
MOVL C00144 BC00144 V=166.7 PL=0
REFP 3 C00145 BC00145
CALL JOB:SEARCH-R1
SET P0355 P0006
SFTON P0355
MOVL C00146 BC00146 V=166.7 PL=0
SFTOF
'------------------------
'W253A L
'------------------------
MOVJ C00147 BC00147 VJ=40.00
MOVL C00148 BC00148 V=166.7 PL=0
REFP 3 C00149 BC00149
CALL JOB:SEARCH-R1
SET P0356 P0006
SFTON P0356
MOVL C00150 BC00150 V=166.7 PL=0
REFP 3 C00151 BC00151
CALL JOB:SEARCH-R1
SET P0356 P0006
SFTON P0356
MOVL C00152 BC00152 V=166.7 PL=0
SFTOF
'------------------------
'W256A P
'------------------------
MOVJ C00153 BC00153 VJ=40.00
MOVL C00154 BC00154 V=166.7 PL=0
REFP 3 C00155 BC00155
CALL JOB:SEARCH-R1
SET P0357 P0006
SFTON P0357
MOVL C00156 BC00156 V=166.7 PL=0
REFP 3 C00157 BC00157
CALL JOB:SEARCH-R1
SET P0357 P0006
SFTON P0357
MOVL C00158 BC00158 V=166.7 PL=0
SFTOF
'------------------------
'W256A L
'------------------------
MOVJ C00159 BC00159 VJ=40.00
MOVL C00160 BC00160 V=166.7 PL=0
REFP 3 C00161 BC00161
CALL JOB:SEARCH-R1
SET P0358 P0006
SFTON P0358
MOVL C00162 BC00162 V=166.7 PL=0
REFP 3 C00163 BC00163
CALL JOB:SEARCH-R1
SET P0358 P0006
SFTON P0358
MOVL C00164 BC00164 V=166.7 PL=0
SFTOF
'------------------------
'W252A P
'------------------------
MOVL C00165 BC00165 V=666.7
MOVL C00166 BC00166 V=166.7 PL=0
REFP 3 C00167 BC00167
CALL JOB:SEARCH-R1
SET P0359 P0006
SFTON P0359
MOVL C00168 BC00168 V=166.7 PL=0
REFP 3 C00169 BC00169
CALL JOB:SEARCH-R1
SET P0359 P0006
SFTON P0359
MOVL C00170 BC00170 V=166.7 PL=0
SFTOF
'------------------------
'W252A L
'------------------------
MOVL C00171 BC00171 V=500.0
MOVL C00172 BC00172 V=166.7 PL=0
REFP 3 C00173 BC00173
CALL JOB:SEARCH-R1
SET P0360 P0006
SFTON P0360
MOVL C00174 BC00174 V=166.7 PL=0
REFP 3 C00175 BC00175
CALL JOB:SEARCH-R1
SET P0360 P0006
SFTON P0360
MOVL C00176 BC00176 V=166.7 PL=0
SFTOF
'------------------------
'W255A
'------------------------
MOVL C00177 BC00177 V=500.0
MOVL C00178 BC00178 V=166.7 PL=0
REFP 3 C00179 BC00179
CALL JOB:SEARCH-R1
SET P0361 P0006
SFTON P0361
MOVL C00180 BC00180 V=166.7 PL=0
REFP 3 C00181 BC00181
CALL JOB:SEARCH-R1
SET P0361 P0006
SFTON P0361
MOVL C00182 BC00182 V=166.7 PL=0
SFTOF
MOVL C00183 BC00183 V=666.7
MOVL C00184 BC00184 V=666.7
MOVL C00185 BC00185 V=666.7
MOVJ C00186 BC00186 VJ=40.00
MOVJ C00187 BC00187 VJ=40.00
MOVJ C00188 BC00188 VJ=40.00
COMM MOVJ C00189 BC00189 VJ=40.00
COMM MOVJ C00190 BC00190 VJ=40.00
COMM MOVJ C00191 BC00191 VJ=40.00
COMM MOVJ C00192 BC00192 VJ=40.00
COMM MOVJ C00193 BC00193 VJ=30.00
COMM '------------------------
COMM 'W61.3
COMM '------------------------
COMM MOVL C00194 BC00194 V=500.0
COMM MOVL C00195 BC00195 V=166.7 PL=0
COMM REFP 3 C00196 BC00196
COMM CALL JOB:SEARCH-R1
COMM SET P0400 P0006
COMM SFTON P0400
COMM MOVL C00197 BC00197 V=166.7 PL=0
COMM REFP 3 C00198 BC00198
COMM CALL JOB:SEARCH-R1
COMM SET P0400 P0006
COMM SFTON P0400
COMM MOVL C00199 BC00199 V=166.7 PL=0
COMM SFTOF
COMM 'BELKA PRZEJAZD
COMM MOVL C00200 BC00200 V=333.3
COMM '------------------------
COMM 'W61.5
COMM '------------------------
COMM MOVL C00201 BC00201 V=166.7 PL=0
COMM REFP 3 C00202 BC00202
COMM CALL JOB:SEARCH-R1
COMM SET P0401 P0006
COMM SFTON P0401
COMM MOVL C00203 BC00203 V=166.7 PL=0
COMM REFP 3 C00204 BC00204
COMM CALL JOB:SEARCH-R1
COMM SET P0401 P0006
COMM SFTON P0401
COMM MOVL C00205 BC00205 V=166.7 PL=0
COMM SFTOF
COMM '------------------------
COMM 'W61.7
COMM '------------------------
COMM MOVL C00206 BC00206 V=500.0
COMM MOVL C00207 BC00207 V=166.7 PL=0
COMM REFP 3 C00208 BC00208
COMM CALL JOB:SEARCH-R1
COMM SET P0402 P0006
COMM SFTON P0402
COMM MOVL C00209 BC00209 V=166.7 PL=0
COMM REFP 3 C00210 BC00210
COMM CALL JOB:SEARCH-R1
COMM SET P0402 P0006
COMM SFTON P0402
COMM MOVL C00211 BC00211 V=166.7 PL=0
COMM SFTOF
COMM MOVL C00212 BC00212 V=500.0
COMM '------------------------
COMM 'W61.10
COMM '------------------------
COMM MOVJ C00213 BC00213 VJ=30.00
COMM MOVJ C00214 BC00214 VJ=50.00
COMM MOVJ C00215 BC00215 VJ=50.00
COMM MOVL C00216 BC00216 V=500.0
COMM MOVL C00217 BC00217 V=166.7 PL=0
COMM REFP 3 C00218 BC00218
COMM CALL JOB:SEARCH-R1
COMM SET P0403 P0006
COMM SFTON P0403
COMM MOVL C00219 BC00219 V=166.7 PL=0
COMM REFP 3 C00220 BC00220
COMM CALL JOB:SEARCH-R1
COMM SET P0403 P0006
COMM SFTON P0403
COMM MOVL C00221 BC00221 V=166.7 PL=0
COMM SFTOF
COMM MOVL C00222 BC00222 V=333.3
COMM '------------------------
COMM 'W61.12
COMM '------------------------
COMM MOVL C00223 BC00223 V=666.7
COMM MOVL C00224 BC00224 V=166.7 PL=0
COMM REFP 3 C00225 BC00225
COMM CALL JOB:SEARCH-R1
COMM SET P0404 P0006
COMM SFTON P0404
COMM MOVL C00226 BC00226 V=166.7 PL=0
COMM REFP 3 C00227 BC00227
COMM CALL JOB:SEARCH-R1
COMM SET P0404 P0006
COMM SFTON P0404
COMM MOVL C00228 BC00228 V=166.7 PL=0
COMM SFTOF
COMM '------------------------
COMM 'W61.15
COMM '------------------------
COMM MOVL C00229 BC00229 V=666.7
COMM MOVL C00230 BC00230 V=166.7 PL=0
COMM REFP 3 C00231 BC00231
COMM CALL JOB:SEARCH-R1
COMM SET P0405 P0006
COMM SFTON P0405
COMM MOVL C00232 BC00232 V=166.7 PL=0
COMM REFP 3 C00233 BC00233
COMM CALL JOB:SEARCH-R1
COMM SET P0405 P0006
COMM SFTON P0405
COMM MOVL C00234 BC00234 V=166.7 PL=0
COMM SFTOF
COMM MOVL C00235 BC00235 V=666.7
COMM MOVJ C00236 BC00236 VJ=50.00
COMM MOVJ C00237 BC00237 VJ=50.00
COMM MOVJ C00238 BC00238 VJ=50.00
COMM '------------------------
COMM 'W61.17
COMM '------------------------
COMM MOVL C00239 BC00239 V=416.7
COMM MOVL C00240 BC00240 V=166.7 PL=0
COMM REFP 3 C00241 BC00241
COMM CALL JOB:SEARCH-R1
COMM SET P0406 P0006
COMM SFTON P0406
COMM MOVL C00242 BC00242 V=166.7 PL=0
COMM REFP 3 C00243 BC00243
COMM CALL JOB:SEARCH-R1
COMM SET P0406 P0006
COMM SFTON P0406
COMM MOVL C00244 BC00244 V=166.7 PL=0
COMM SFTOF
COMM MOVL C00245 BC00245 V=333.3
COMM '------------------------
COMM 'W61.20
COMM '------------------------
COMM MOVL C00246 BC00246 V=666.7
COMM MOVL C00247 BC00247 V=166.7 PL=0
COMM REFP 3 C00248 BC00248
COMM CALL JOB:SEARCH-R1
COMM SET P0407 P0006
COMM SFTON P0407
COMM MOVL C00249 BC00249 V=166.7 PL=0
COMM REFP 3 C00250 BC00250
COMM CALL JOB:SEARCH-R1
COMM SET P0407 P0006
COMM SFTON P0407
COMM MOVL C00251 BC00251 V=166.7 PL=0
COMM SFTOF
COMM '------------------------
COMM 'W61.23
COMM '------------------------
COMM MOVL C00252 BC00252 V=500.0
COMM MOVL C00253 BC00253 V=166.7 PL=0
COMM REFP 3 C00254 BC00254
COMM CALL JOB:SEARCH-R1
COMM SET P0408 P0006
COMM SFTON P0408
COMM MOVL C00255 BC00255 V=166.7 PL=0
COMM REFP 3 C00256 BC00256
COMM CALL JOB:SEARCH-R1
COMM SET P0408 P0006
COMM SFTON P0408
COMM MOVL C00257 BC00257 V=166.7 PL=0
COMM SFTOF
COMM MOVL C00258 BC00258 V=333.3
COMM MOVL C00259 BC00259 V=666.7
COMM MOVL C00260 BC00260 V=666.7
COMM '------------------------
COMM 'W61.25
COMM '------------------------
COMM MOVL C00261 BC00261 V=500.0
COMM MOVL C00262 BC00262 V=166.7 PL=0
COMM REFP 3 C00263 BC00263
COMM CALL JOB:SEARCH-R1
COMM SET P0409 P0006
COMM SFTON P0409
COMM MOVL C00264 BC00264 V=166.7 PL=0
COMM REFP 3 C00265 BC00265
COMM CALL JOB:SEARCH-R1
COMM SET P0409 P0006
COMM SFTON P0409
COMM MOVL C00266 BC00266 V=166.7 PL=0
COMM SFTOF
COMM MOVL C00267 BC00267 V=666.7
COMM MOVJ C00268 BC00268 VJ=50.00
COMM MOVJ C00269 BC00269 VJ=50.00
COMM GETE D040 P0409 (1)
COMM GETE D041 P0409 (2)
COMM GETE D042 P0409 (3)
COMM SETE P0410 (1) D040
COMM SETE P0410 (2) D041
COMM SETE P0410 (3) D042
COMM '------------------------
COMM 'W61.30
COMM '------------------------
COMM MOVL C00270 BC00270 V=500.0
COMM MOVL C00271 BC00271 V=166.7 PL=0
COMM REFP 3 C00272 BC00272
COMM CALL JOB:SEARCH-R1
COMM SET P0411 P0006
COMM SFTON P0411
COMM MOVL C00273 BC00273 V=166.7 PL=0
COMM REFP 3 C00274 BC00274
COMM CALL JOB:SEARCH-R1
COMM SET P0411 P0006
COMM SFTON P0411
COMM MOVL C00275 BC00275 V=166.7 PL=0
COMM SFTOF
COMM MOVL C00276 BC00276 V=666.7
COMM MOVJ C00277 BC00277 VJ=50.00
MOVJ C00278 BC00278 VJ=50.00
CALL JOB:FRONT_SEARCH_-90ST-2_4690
MOVJ C00279 BC00279 VJ=60.00
MOVJ C00280 BC00280 VJ=50.00
MOVJ C00281 BC00281 VJ=50.00
MOVL C00282 BC00282 V=666.7
MOVJ C00283 BC00283 VJ=30.00
'------------------------
'W65.3
'------------------------
SFTON P0300
MOVL C00284 BC00284 V=333.3
MOVL C00285 BC00285 V=166.7 PL=0
MACRO1 MJ#(0) ARGF30
ARCON
MOVL C00286 BC00286 V=11.7
ARCOF
MOVL C00287 BC00287 V=166.7
SFTOF
'------------------------
'W65.5
'------------------------
SFTON P0301
MOVL C00288 BC00288 V=666.7
MOVL C00289 BC00289 V=166.7 PL=0
MACRO1 MJ#(0) ARGF29
ARCON
MOVL C00290 BC00290 V=11.7
ARCOF
MOVL C00291 BC00291 V=166.7
SFTOF
MOVL C00292 BC00292 V=500.0
MOVL C00293 BC00293 V=666.7
MOVJ C00294 BC00294 VJ=40.00
COMM MOVJ C00295 BC00295 VJ=60.00
COMM '::::::::::::::::::::::::::::::::
COMM '::::::::::::::::::::::::::::::::
COMM '::::::::::::::::::::::::::::::::
COMM '::::::::::::::::::::::::::::::::
COMM '::::::::::::::::::::::::::::::::
COMM MOVJ C00296 BC00296 VJ=50.00
COMM MOVJ C00297 BC00297 VJ=50.00
COMM MOVJ C00298 BC00298 VJ=40.00
COMM MOVJ C00299 BC00299 VJ=40.00
COMM MOVJ C00300 BC00300 VJ=40.00
COMM MOVJ C00301 BC00301 VJ=40.00
COMM MOVL C00302 BC00302 V=666.7
COMM '------------------------
COMM 'W61.3
COMM '------------------------
COMM SFTON P0400
COMM ARCOF
COMM MOVL C00303 BC00303 V=500.0
COMM SFTOF
COMM 'BELKA PRZEJAZD
COMM '------------------------
COMM 'W61.5
COMM '------------------------
COMM SFTON P0401
COMM MOVL C00304 BC00304 V=666.7
COMM MOVL C00305 BC00305 V=166.7 PL=0
COMM MACRO1 MJ#(0) ARGF24
COMM ARCON
COMM MOVL C00306 BC00306 V=7.5
COMM ARCOF
COMM MOVL C00307 BC00307 V=250.0
COMM SFTOF
COMM MOVL C00308 BC00308 V=500.0
COMM MOVJ C00309 BC00309 VJ=40.00
COMM MOVJ C00310 BC00310 VJ=40.00
COMM MOVJ C00311 BC00311 VJ=50.00
COMM MOVJ C00312 BC00312 VJ=50.00
MOVJ C00313 BC00313 VJ=50.00
MOVJ C00314 BC00314 VJ=50.00
MOVL C00315 BC00315 V=666.7
'------------------------
'W250A
'------------------------
SFTON P0354
MOVL C00316 BC00316 V=666.7
MOVL C00317 BC00317 V=166.7 PL=0
MACRO1 MJ#(0) ARGF29
ARCON
SFTOF
SFTON P0353
MOVL C00318 BC00318 V=12.5
ARCOF
MOVL C00319 BC00319 V=333.3
SFTOF
MOVJ C00320 BC00320 VJ=50.00
MOVJ C00321 BC00321 VJ=60.00
MOVJ C00322 BC00322 VJ=40.00
MOVJ C00323 BC00323 VJ=50.00
MOVJ C00324 BC00324 VJ=40.00
MOVJ C00325 BC00325 VJ=30.00
MOVJ C00326 BC00326 VJ=15.00
'------------------------
'W65.7
'------------------------
SFTON P0302
MOVL C00327 BC00327 V=833.3
MOVL C00328 BC00328 V=166.7 PL=0
MACRO1 MJ#(0) ARGF30
ARCON
MOVL C00329 BC00329 V=11.7
ARCOF
MOVL C00330 BC00330 V=166.7
SFTOF
'------------------------
'W65.10
'------------------------
SFTON P0303
MOVL C00331 BC00331 V=666.7
MOVL C00332 BC00332 V=166.7 PL=0
ARCON
MOVL C00333 BC00333 V=11.7
ARCOF
MOVL C00334 BC00334 V=166.7
SFTOF
COMM MOVL C00335 BC00335 V=333.3
COMM MOVL C00336 BC00336 V=333.3
COMM MOVJ C00337 BC00337 VJ=30.00
COMM MOVJ C00338 BC00338 VJ=30.00
COMM MOVJ C00339 BC00339 VJ=50.00
COMM '::::::::::::::::::::::::::::::::
COMM '::::::::::::::::::::::::::::::::
COMM '------------------------
COMM 'W61.7
COMM '------------------------
COMM '::::::::::::::::::::::::::::::::
COMM '::::::::::::::::::::::::::::::::
COMM MOVJ C00340 BC00340 VJ=30.00
COMM MOVJ C00341 BC00341 VJ=30.00
COMM MOVJ C00342 BC00342 VJ=40.00
COMM SFTON P0402
COMM MOVL C00343 BC00343 V=500.0
COMM MOVL C00344 BC00344 V=166.7 PL=0
COMM MACRO1 MJ#(0) ARGF24
COMM ARCON
COMM MOVL C00345 BC00345 V=7.5
COMM ARCOF
COMM MOVL C00346 BC00346 V=250.0
COMM SFTOF
COMM MOVJ C00347 BC00347 VJ=30.00
COMM MOVJ C00348 BC00348 VJ=40.00
COMM MOVJ C00349 BC00349 VJ=50.00
COMM '------------------------
COMM 'W61.10
COMM '------------------------
COMM SFTON P0403
COMM MOVL C00350 BC00350 V=500.0
COMM MOVL C00351 BC00351 V=166.7 PL=0
COMM MACRO1 MJ#(0) ARGF24
COMM ARCON
COMM MOVL C00352 BC00352 V=7.5
COMM ARCOF
COMM MOVL C00353 BC00353 V=250.0
COMM SFTOF
COMM MOVL C00354 BC00354 V=500.0
COMM MOVL C00355 BC00355 V=666.7
COMM MOVL C00356 BC00356 V=666.7
COMM MOVJ C00357 BC00357 VJ=50.00
COMM MOVJ C00358 BC00358 VJ=50.00
COMM MOVJ C00359 BC00359 VJ=50.00
COMM '::::::::::::::::::::::::
COMM '::::::::::::::::::::::::
COMM '::::::::::::::::::::::::
COMM '::::::::::::::::::::::::
COMM '::::::::::::::::::::::::
COMM '::::::::::::::::::::::::
COMM '::::::::::::::::::::::::
COMM MOVJ C00360 BC00360 VJ=50.00
COMM MOVJ C00361 BC00361 VJ=50.00
COMM MOVJ C00362 BC00362 VJ=50.00
COMM '------------------------
COMM 'W251B
COMM '------------------------
COMM MOVL C00363 BC00363 V=500.0
COMM MOVL C00364 BC00364 V=500.0
COMM SFTON P0350
COMM MOVL C00365 BC00365 V=166.7 PL=0
COMM MACRO1 MJ#(0) ARGF9
COMM ARCON
COMM SFTOF
COMM SFTON P0350
COMM MOVL C00366 BC00366 V=11.3
COMM MOVL C00367 BC00367 V=11.3
COMM ARCOF
COMM MOVL C00368 BC00368 V=333.3
COMM SFTOF
COMM MOVJ C00369 BC00369 VJ=50.00
COMM MOVJ C00370 BC00370 VJ=50.00
COMM MOVJ C00371 BC00371 VJ=10.00
COMM MOVJ C00372 BC00372 VJ=50.00
COMM MOVJ C00373 BC00373 VJ=50.00
COMM MOVJ C00374 BC00374 VJ=25.00
COMM MOVJ C00375 BC00375 VJ=20.00
COMM MOVJ C00376 BC00376 VJ=20.00
'------------------------
'W65.12
'------------------------
SFTON P0304
MOVL C00377 BC00377 V=333.3
MOVL C00378 BC00378 V=166.7 PL=0
MACRO1 MJ#(0) ARGF30
ARCON
MOVL C00379 BC00379 V=11.7
ARCOF
MOVL C00380 BC00380 V=166.7
SFTOF
'------------------------
'W65.15
'------------------------
MOVL C00381 BC00381 V=250.0
MOVL C00382 BC00382 V=416.7
MOVL C00383 BC00383 V=666.7
COMM MOVJ C00384 BC00384 VJ=50.00
COMM MOVJ C00385 BC00385 VJ=50.00
COMM '::::::::::::::::::::::::
COMM '::::::::::::::::::::::::
COMM '::::::::::::::::::::::::
COMM '::::::::::::::::::::::::
COMM '::::::::::::::::::::::::
COMM '::::::::::::::::::::::::
COMM '::::::::::::::::::::::::
COMM MOVJ C00386 BC00386 VJ=50.00
COMM MOVJ C00387 BC00387 VJ=50.00
COMM MOVJ C00388 BC00388 VJ=50.00
COMM '::::::::::::::::::::::::::::::::
COMM '::::::::::::::::::::::::::::::::
COMM '------------------------
COMM 'W61.12
COMM '------------------------
COMM '::::::::::::::::::::::::::::::::
COMM '::::::::::::::::::::::::::::::::
COMM MOVL C00389 BC00389 V=833.3
COMM MOVL C00390 BC00390 V=666.7
COMM MOVL C00391 BC00391 V=500.0
COMM SFTON P0404
COMM MOVL C00392 BC00392 V=166.7 PL=0
COMM MACRO1 MJ#(0) ARGF24
COMM ARCON
COMM MOVL C00393 BC00393 V=6.7
COMM ARCOF
COMM MOVL C00394 BC00394 V=333.3
COMM SFTOF
COMM MOVL C00395 BC00395 V=500.0
COMM MOVL C00396 BC00396 V=666.7
COMM '------------------------
COMM 'W61.15
COMM '------------------------
COMM SFTON P0405
COMM MOVL C00397 BC00397 V=666.7
COMM MOVL C00398 BC00398 V=166.7 PL=0
COMM MACRO1 MJ#(0) ARGF24
COMM ARCON
COMM MOVL C00399 BC00399 V=6.7
COMM ARCOF
COMM MOVL C00400 BC00400 V=250.0
COMM SFTOF
COMM MOVJ C00401 BC00401 VJ=40.00
COMM MOVJ C00402 BC00402 VJ=40.00
COMM MOVJ C00403 BC00403 VJ=40.00
COMM MOVJ C00404 BC00404 VJ=40.00
COMM '::::::::::::::::::::::::
COMM '::::::::::::::::::::::::
COMM '::::::::::::::::::::::::
COMM '::::::::::::::::::::::::
COMM '::::::::::::::::::::::::
COMM '::::::::::::::::::::::::
COMM '::::::::::::::::::::::::
COMM MOVJ C00405 BC00405 VJ=40.00
COMM MOVJ C00406 BC00406 VJ=40.00
COMM '------------------------
COMM 'W252B
COMM '------------------------
SFTON P0359
MOVL C00407 BC00407 V=666.7
MOVL C00408 BC00408 V=166.7 PL=0
MACRO1 MJ#(0) ARGF29
ARCON
SFTOF
SFTON P0358
MOVL C00409 BC00409 V=11.7
ARCOF
MOVL C00410 BC00410 V=250.0
SFTOF
MOVJ C00411 BC00411 VJ=50.00
MOVJ C00412 BC00412 VJ=50.00
MOVJ C00413 BC00413 VJ=60.00
MOVJ C00414 BC00414 VJ=40.00
MOVJ C00415 BC00415 VJ=30.00
MOVL C00416 BC00416 V=500.0
MOVL C00417 BC00417 V=333.3
'------------------------
'W65.17
'------------------------
MOVL C00418 BC00418 V=333.3
SFTON P0306
MOVL C00419 BC00419 V=166.7 PL=0
MACRO1 MJ#(0) ARGF30
ARCON
MOVL C00420 BC00420 V=11.7
ARCOF
MOVL C00421 BC00421 V=166.7
SFTOF
MOVL C00422 BC00422 V=333.3
MOVL C00423 BC00423 V=500.0
MOVJ C00424 BC00424 VJ=40.00
COMM MOVJ C00425 BC00425 VJ=60.00
COMM MOVJ C00426 BC00426 VJ=60.00
COMM '::::::::::::::::::::::::
COMM '::::::::::::::::::::::::
COMM '::::::::::::::::::::::::
COMM '::::::::::::::::::::::::
COMM '::::::::::::::::::::::::
COMM '::::::::::::::::::::::::
COMM '::::::::::::::::::::::::
COMM MOVJ C00427 BC00427 VJ=60.00
COMM '::::::::::::::::::::::::::::::::
COMM '::::::::::::::::::::::::::::::::
COMM '------------------------
COMM 'W61.17
COMM '------------------------
COMM '::::::::::::::::::::::::::::::::
COMM '::::::::::::::::::::::::::::::::
COMM SFTON P0406
COMM MOVJ C00428 BC00428 VJ=40.00
COMM MOVL C00429 BC00429 V=500.0
COMM MOVL C00430 BC00430 V=166.7 PL=0
COMM MACRO1 MJ#(0) ARGF24
COMM ARCON
COMM MOVL C00431 BC00431 V=6.7
COMM ARCOF
COMM MOVL C00432 BC00432 V=333.3
COMM SFTOF
COMM MOVJ C00433 BC00433 VJ=30.00
COMM MOVJ C00434 BC00434 VJ=40.00
COMM MOVJ C00435 BC00435 VJ=50.00
COMM '------------------------
COMM 'W253A
'------------------------
COMM MOVJ C00436 BC00436 VJ=50.00
MOVJ C00437 BC00437 VJ=50.00
SFTON P0356
MOVL C00438 BC00438 V=500.0
MOVL C00439 BC00439 V=500.0
MOVL C00440 BC00440 V=166.7 PL=0
MACRO1 MJ#(0) ARGF29
ARCON
SFTOF
SFTON P0355
MOVL C00441 BC00441 V=12.5
ARCOF
MOVL C00442 BC00442 V=333.3
SFTOF
MOVJ C00443 BC00443 VJ=50.00
MOVJ C00444 BC00444 VJ=50.00
MOVJ C00445 BC00445 VJ=50.00
MOVJ C00446 BC00446 VJ=50.00
MOVJ C00447 BC00447 VJ=50.00
MOVJ C00448 BC00448 VJ=50.00
MOVJ C00449 BC00449 VJ=40.00
MOVL C00450 BC00450 V=333.3
'------------------------
'W65.20
'------------------------
SFTON P0307
MOVL C00451 BC00451 V=500.0
MOVL C00452 BC00452 V=333.3
MOVL C00453 BC00453 V=166.7 PL=0
MACRO1 MJ#(0) ARGF30
ARCON
MOVL C00454 BC00454 V=11.7
ARCOF
MOVL C00455 BC00455 V=250.0
SFTOF
MOVL C00456 BC00456 V=666.7
MOVL C00457 BC00457 V=333.3
MOVL C00458 BC00458 V=500.0
MOVL C00459 BC00459 V=500.0
MOVJ C00460 BC00460 VJ=50.00
COMM MOVJ C00461 BC00461 VJ=50.00
COMM MOVJ C00462 BC00462 VJ=50.00
COMM MOVJ C00463 BC00463 VJ=50.00
COMM '::::::::::::::::::::::::
COMM '::::::::::::::::::::::::
COMM '::::::::::::::::::::::::
COMM '::::::::::::::::::::::::
COMM '::::::::::::::::::::::::
COMM '::::::::::::::::::::::::
COMM '::::::::::::::::::::::::
COMM MOVJ C00464 BC00464 VJ=40.00
COMM MOVJ C00465 BC00465 VJ=40.00
COMM '::::::::::::::::::::::::::::::::
COMM '::::::::::::::::::::::::::::::::
COMM '------------------------
COMM 'W61.20
COMM '------------------------
COMM '::::::::::::::::::::::::::::::::
COMM '::::::::::::::::::::::::::::::::
COMM SFTON P0407
COMM MOVL C00466 BC00466 V=666.7
COMM MOVL C00467 BC00467 V=333.3
COMM MOVL C00468 BC00468 V=166.7 PL=0
COMM MACRO1 MJ#(0) ARGF24
COMM ARCON
COMM MOVL C00469 BC00469 V=6.7
COMM ARCOF
COMM MOVL C00470 BC00470 V=250.0
COMM SFTOF
COMM '::::::::::::::::::::::::
COMM '::::::::::::::::::::::::
COMM '::::::::::::::::::::::::
COMM '::::::::::::::::::::::::
COMM '::::::::::::::::::::::::
COMM MOVL C00471 BC00471 V=500.0
COMM MOVJ C00472 BC00472 VJ=50.00
COMM MOVJ C00473 BC00473 VJ=50.00
COMM MOVJ C00474 BC00474 VJ=50.00
COMM '------------------------
COMM 'W254A
COMM '------------------------
COMM MOVJ C00475 BC00475 VJ=50.00
MOVJ C00476 BC00476 VJ=50.00
SFTON P0352
MOVL C00477 BC00477 V=666.7
MOVL C00478 BC00478 V=500.0
MOVL C00479 BC00479 V=250.0 PL=0
MACRO1 MJ#(0) ARGF29
ARCON
SFTOF
SFTON P0351
MOVL C00480 BC00480 V=12.5
ARCOF
MOVL C00481 BC00481 V=333.3
MOVL C00482 BC00482 V=666.7
SFTOF
COMM MOVJ C00483 BC00483 VJ=50.00
COMM MOVJ C00484 BC00484 VJ=80.00
COMM MOVJ C00485 BC00485 VJ=50.00
MOVJ C00486 BC00486 VJ=50.00
MOVJ C00487 BC00487 VJ=30.00
MOVJ C00488 BC00488 VJ=30.00
MOVJ C00489 BC00489 VJ=20.00
MOVL C00490 BC00490 V=666.7
'------------------------
'W65.23
'------------------------
MOVL C00491 BC00491 V=333.3
MOVL C00492 BC00492 V=166.7
SFTON P0308
MOVL C00493 BC00493 V=166.7 PL=0
MACRO1 MJ#(0) ARGF30
ARCON
MOVL C00494 BC00494 V=11.7
ARCOF
MOVL C00495 BC00495 V=250.0
SFTOF
'------------------------
'W65.25
'------------------------
COMM SFTON P0309
COMM MOVL C00496 BC00496 V=166.7
COMM MOVL C00497 BC00497 V=166.7 PL=0
COMM ARCON
COMM MOVL C00498 BC00498 V=11.7
COMM ARCOF
COMM MOVL C00499 BC00499 V=250.0
COMM SFTOF
MOVL C00500 BC00500 V=500.0
MOVL C00501 BC00501 V=666.7
MOVL C00502 BC00502 V=666.7
MOVJ C00503 BC00503 VJ=40.00
MOVJ C00504 BC00504 VJ=40.00
MOVJ C00505 BC00505 VJ=50.00
COMM '::::::::::::::::::::::::
COMM '::::::::::::::::::::::::
COMM '::::::::::::::::::::::::
COMM '::::::::::::::::::::::::
COMM '::::::::::::::::::::::::
COMM '::::::::::::::::::::::::
COMM '::::::::::::::::::::::::
COMM MOVJ C00506 BC00506 VJ=50.00
COMM MOVJ C00507 BC00507 VJ=50.00
COMM MOVJ C00508 BC00508 VJ=50.00
COMM '::::::::::::::::::::::::::::::::
COMM '::::::::::::::::::::::::::::::::
COMM '------------------------
COMM 'W61.23
COMM '------------------------
COMM '::::::::::::::::::::::::::::::::
COMM '::::::::::::::::::::::::::::::::
COMM SFTON P0408
COMM MOVL C00509 BC00509 V=500.0
COMM MOVL C00510 BC00510 V=666.7
COMM MOVL C00511 BC00511 V=166.7 PL=0
COMM MACRO1 MJ#(0) ARGF24
COMM ARCON
COMM MOVL C00512 BC00512 V=8.3
COMM ARCOF
COMM MOVL C00513 BC00513 V=250.0
COMM SFTOF
COMM MOVL C00514 BC00514 V=666.7
COMM '------------------------
COMM 'W61.25
COMM '------------------------
COMM SFTON P0409
COMM MOVL C00515 BC00515 V=500.0
COMM MOVL C00516 BC00516 V=166.7 PL=0
COMM MACRO1 MJ#(0) ARGF24
COMM ARCON
COMM MOVL C00517 BC00517 V=8.3
COMM ARCOF
COMM MOVL C00518 BC00518 V=166.7
COMM SFTOF
COMM MOVL C00519 BC00519 V=500.0
COMM MOVJ C00520 BC00520 VJ=20.00
COMM '::::::::::::::::::::::::
COMM '::::::::::::::::::::::::
COMM '::::::::::::::::::::::::
COMM '::::::::::::::::::::::::
COMM '::::::::::::::::::::::::
COMM MOVJ C00521 BC00521 VJ=50.00
COMM MOVJ C00522 BC00522 VJ=50.00
MOVJ C00523 BC00523 VJ=40.00
'------------------------
'W255A
MOVL C00524 BC00524 V=500.0
MOVL C00525 BC00525 V=666.7
SFTON P0361
MOVL C00526 BC00526 V=166.7 PL=0
MACRO1 MJ#(0) ARGF29
ARCON
MOVL C00527 BC00527 V=12.5
ARCOF
MOVL C00528 BC00528 V=333.3
SFTOF
MOVL C00529 BC00529 V=666.7
MOVL C00530 BC00530 V=666.7
MOVL C00531 BC00531 V=666.7
MOVJ C00532 BC00532 VJ=50.00
MOVJ C00533 BC00533 VJ=70.00
MOVJ C00534 BC00534 VJ=70.00
MOVJ C00535 BC00535 VJ=50.00
MOVJ C00536 BC00536 VJ=50.00
MOVJ C00537 BC00537 VJ=50.00
MOVL C00538 BC00538 V=500.0
'------------------------
'W31.28
'------------------------
SFTON P0310
MOVL C00539 BC00539 V=333.3
COMM MOVL C00540 BC00540 V=333.3
COMM MOVL C00541 BC00541 V=333.3
COMM MACRO1 MJ#(0) ARGF10
COMM MOVL C00542 BC00542 V=166.7
COMM ARCON
COMM MOVL C00543 BC00543 V=10.8
COMM ARCOF
MACRO1 MJ#(0) ARGF30
MOVL C00544 BC00544 V=200.0
ARCON
MOVL C00545 BC00545 V=11.7
ARCOF
MOVL C00546 BC00546 V=166.7
SFTOF
'------------------------
COMM 'W31.30
COMM '------------------------
COMM SFTON P0311
COMM MOVL C00547 BC00547 V=333.3
COMM MOVL C00548 BC00548 V=166.7 PL=0
COMM MACRO1 MJ#(0) ARGF9
COMM ARCON
COMM MOVL C00549 BC00549 V=10.8
COMM ARCOF
COMM MOVL C00550 BC00550 V=250.0
COMM SFTOF
MOVL C00551 BC00551 V=166.7
MOVL C00552 BC00552 V=500.0
MOVL C00553 BC00553 V=500.0
MOVL C00554 BC00554 V=666.7
MOVJ C00555 BC00555 VJ=25.00
COMM '::::::::::::::::::::::::
COMM '::::::::::::::::::::::::
COMM '::::::::::::::::::::::::
COMM '::::::::::::::::::::::::
COMM '::::::::::::::::::::::::
COMM '::::::::::::::::::::::::
COMM '::::::::::::::::::::::::
COMM MOVJ C00556 BC00556 VJ=20.00
COMM MOVJ C00557 BC00557 VJ=30.00
COMM '::::::::::::::::::::::::::::::::
COMM '::::::::::::::::::::::::::::::::
COMM '------------------------
COMM 'W61.30
COMM '------------------------
COMM '::::::::::::::::::::::::::::::::
COMM '::::::::::::::::::::::::::::::::
COMM SFTON P0411
COMM MOVL C00558 BC00558 V=500.0
COMM MOVL C00559 BC00559 V=166.7 PL=0
COMM MACRO1 MJ#(0) ARGF24
COMM ARCON
COMM MOVL C00560 BC00560 V=7.5
COMM ARCOF
COMM MOVL C00561 BC00561 V=250.0
COMM MOVL C00562 BC00562 V=500.0
COMM MOVL C00563 BC00563 V=166.7 PL=0
COMM MACRO1 MJ#(0) ARGF24
COMM ARCON
COMM MOVL C00564 BC00564 V=7.5
COMM ARCOF
COMM MOVL C00565 BC00565 V=250.0
COMM SFTOF
COMM MOVL C00566 BC00566 V=500.0
COMM SFTOF
COMM MOVL C00567 BC00567 V=500.0
COMM MOVJ C00568 BC00568 VJ=25.00
MOVJ C00569 BC00569 VJ=50.00
MOVJ C00570 BC00570 VJ=50.00
MOVJ C00571 BC00571 VJ=60.00
'------------------------
'W256A
'------------------------
MOVJ C00572 BC00572 VJ=60.00
MOVJ C00573 BC00573 VJ=60.00
SFTON P0358
MOVL C00574 BC00574 V=666.7
MOVL C00575 BC00575 V=250.0
MOVL C00576 BC00576 V=166.7 PL=0
MACRO1 MJ#(0) ARGF29
ARCON
SFTOF
SFTON P0357
MOVL C00577 BC00577 V=12.5
ARCOF
MOVL C00578 BC00578 V=333.3
SFTOF
MOVJ C00579 BC00579 VJ=50.00
MOVJ C00580 BC00580 VJ=50.00
CALL JOB:FRONT_WELD_-90ST-2_4640
CALL JOB:MOVE_OUT_OF_TUNNEL
END
